FUNCTION_BLOCK fbAwait
VAR
	Timer : Tc2_Standard.TON;
END_VAR

METHOD Delay : BOOL
VAR_INPUT
	Timespan : TIME;
END_VAR
Timer(IN := TRUE, PT := Timespan);

IF Timer.Q THEN
	Timer(IN := FALSE, PT := T#0S);
	Delay := TRUE;
END_IF
END_METHOD

METHOD Sometime : BOOL
VAR_INPUT
END_VAR
Sometime := Delay(T#1S);
END_METHOD

END_FUNCTION_BLOCK

(* stored: Version 1.1.0.1, ProductVersion 3.1.4024.6
   POU fbAwait: Id {5d277946-a10c-0945-26ab-70abcf6da4de}, SpecialFunc None
   Method Delay: Id {43578758-a06a-096b-172c-40034bf4da0a}
   Method Sometime: Id {afcdfa1f-c41f-0605-1d11-0da5aa0754c7} *)
